SUBAPPLICATION Ventilsteuerung_Uebung_009 (* Ticker *)
  (* Standard: 61499-2 *)
  (* Version 1.0, 2023-10-23, franz *)
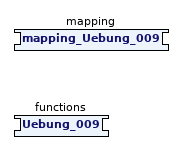
  SUBAPPS
    mapping : mapping_Uebung_009;
    functions : Uebung_009;
  END_SUBAPPS
END_SUBAPPLICATION
